// Mitsubishi GX Works2 project: 241108_PLC_STUDY   PLC: Q02U

PROGRAM MAIN
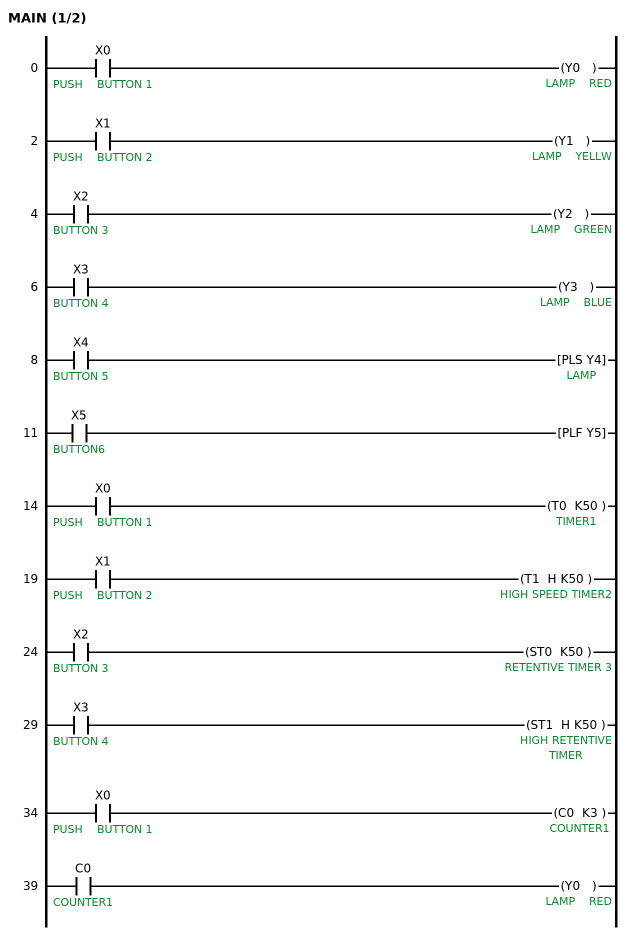
0     LD      X0  ; PUSH    BUTTON 1
      OUT     Y0  ; LAMP    RED
2     LD      X1  ; PUSH    BUTTON 2
      OUT     Y1  ; LAMP    YELLW
4     LD      X2  ; BUTTON 3
      OUT     Y2  ; LAMP    GREEN
6     LD      X3  ; BUTTON 4
      OUT     Y3  ; LAMP    BLUE
8     LD      X4  ; BUTTON 5
      PLS     Y4  ; LAMP
11    LD      X5  ; BUTTON6
      PLF     Y5
14    LD      X0  ; PUSH    BUTTON 1
      OUT     T0 K50  ; TIMER1
19    LD      X1  ; PUSH    BUTTON 2
      OUTH    T1 K50  ; HIGH SPEED TIMER2
24    LD      X2  ; BUTTON 3
      OUT     ST0 K50  ; RETENTIVE TIMER 3
29    LD      X3  ; BUTTON 4
      OUTH    ST1 K50  ; HIGH RETENTIVE TIMER
34    LD      X0  ; PUSH    BUTTON 1
      OUT     C0 K3  ; COUNTER1
39    LD      C0  ; COUNTER1
      OUT     Y0  ; LAMP    RED
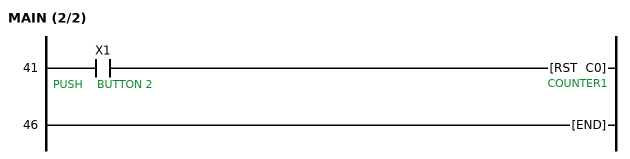
41    LD      X1  ; PUSH    BUTTON 2
      RST     C0  ; COUNTER1
46    END
END_PROGRAM

// device comments not shown above
X6  ; Push    Button 6
X7  ; Push    Button 7
